FUNCTION_BLOCK FB_RollerDoor
VAR_INPUT
    CloseCmd   : BOOL;
    OpenCmd    : BOOL;
END_VAR

VAR_OUTPUT
    CloseOut   : BOOL;
    OpenOut    : BOOL;
    Done       : BOOL;
    Busy       : BOOL;
    ClosedSim  : BOOL;
    OpenedSim  : BOOL;
END_VAR

VAR
    State   : INT := 0;
    tClose  : TON;
    tOpen   : TON;
END_VAR

CASE State OF

0: // Idle
    Done := FALSE;
    Busy := FALSE;
    CloseOut := FALSE;
    OpenOut := FALSE;

    tClose(IN := FALSE);
    tOpen(IN := FALSE);

    IF CloseCmd THEN
        State := 10;
    ELSIF OpenCmd THEN
        State := 20;
    END_IF


10: // Closing
    Busy := TRUE;
    CloseOut := TRUE;

    tClose(IN := TRUE, PT := T#4S);

    IF tClose.Q THEN
        CloseOut := FALSE;
        Busy := FALSE;
        Done := TRUE;
        ClosedSim := TRUE;
        OpenedSim := FALSE;
        tClose(IN := FALSE);
        State := 0;
    END_IF


20: // Opening
    Busy := TRUE;
    OpenOut := TRUE;

    tOpen(IN := TRUE, PT := T#4S);

    IF tOpen.Q THEN
        OpenOut := FALSE;
        Busy := FALSE;
        Done := TRUE;
        OpenedSim := TRUE;
        ClosedSim := FALSE;
        tOpen(IN := FALSE);
        State := 0;
    END_IF

END_CASE

END_FUNCTION_BLOCK

(* stored: Version 1.1.0.1, ProductVersion 3.1.4024.16
   POU FB_RollerDoor: Id {95c47bba-d768-4091-9920-c219f4611596}, SpecialFunc None *)
